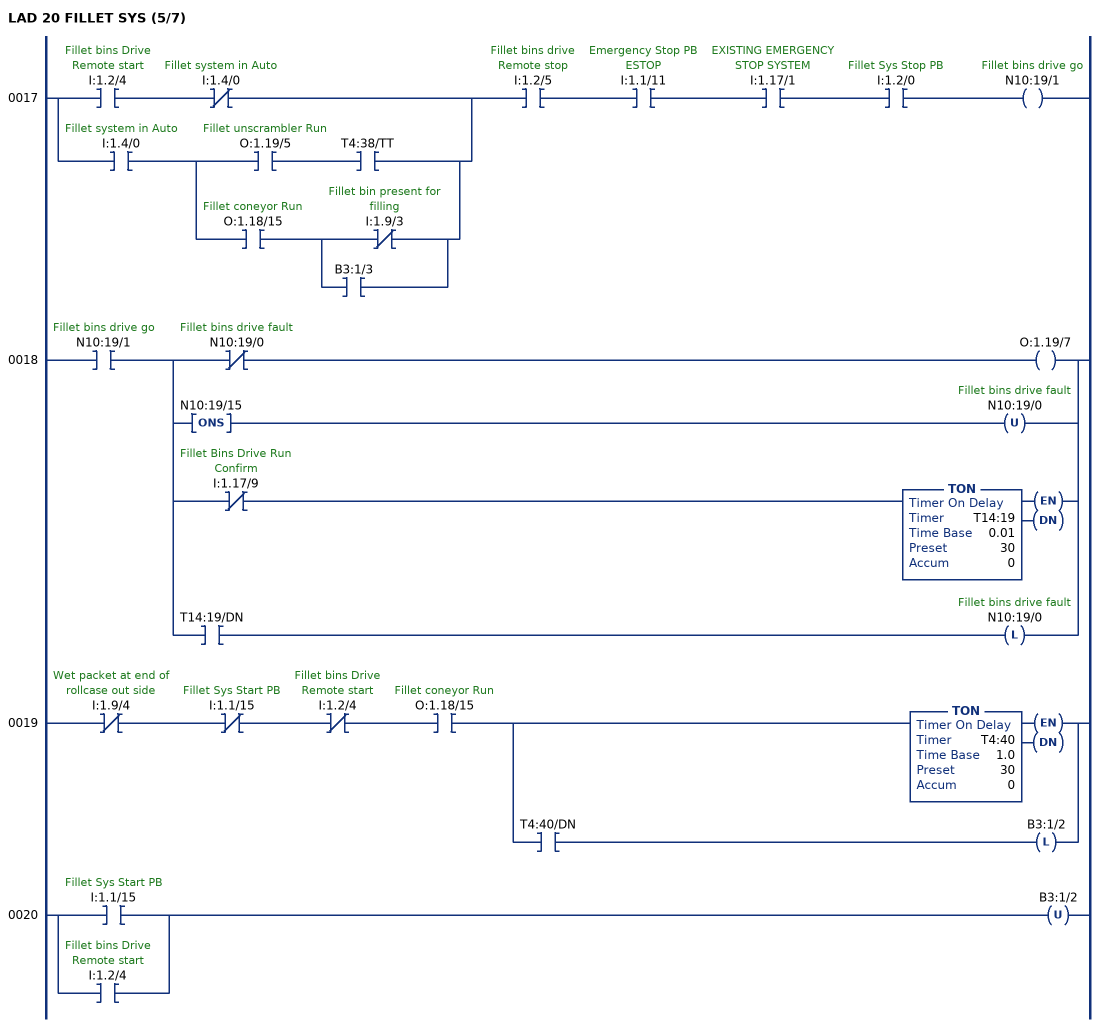
% Rung: 17 %
SOR BST XIC I:1.2/4 XIO I:1.4/0 NXB XIC I:1.4/0 BST XIC O:1.19/5 XIC T4:38/TT NXB XIC O:1.18/15 BST XIO I:1.9/3 NXB XIC B3:1/3 BND BND BND XIC I:1.2/5 XIC I:1.1/11 XIC I:1.17/1 XIC I:1.2/0 OTE N10:19/1 EOR
%   I:1.2/4  "Fillet bins Drive Remote start" %
%   I:1.4/0  "Fillet system in Auto" %
%   O:1.19/5  "Fillet unscrambler Run" %
%   O:1.18/15  "Fillet coneyor Run" %
%   I:1.9/3  "Fillet bin present for filling" %
%   I:1.2/5  "Fillet bins drive Remote stop" %
%   I:1.1/11  ESTOP  "Emergency Stop PB" %
%   I:1.17/1  "EXISTING EMERGENCY STOP SYSTEM" %
%   I:1.2/0  "Fillet Sys Stop PB" %
%   N10:19/1  "Fillet bins drive go" %
% Rung: 18 %
SOR XIC N10:19/1 BST XIO N10:19/0 OTE O:1.19/7 NXB OSR N10:19/15 OTU N10:19/0 NXB XIO I:1.17/9 TON T14:19 0.01 30 0 NXB XIC T14:19/DN OTL N10:19/0 BND EOR
%   N10:19/1  "Fillet bins drive go" %
%   N10:19/0  "Fillet bins drive fault" %
%   I:1.17/9  "Fillet Bins Drive Run Confirm" %
% Rung: 19 %
SOR XIO I:1.9/4 XIO I:1.1/15 XIO I:1.2/4 XIC O:1.18/15 BST TON T4:40 1.0 30 0 NXB XIC T4:40/DN OTL B3:1/2 BND EOR
%   I:1.9/4  "Wet packet at end of rollcase out side" %
%   I:1.1/15  "Fillet Sys Start PB" %
%   I:1.2/4  "Fillet bins Drive Remote start" %
%   O:1.18/15  "Fillet coneyor Run" %
% Rung: 20 %
SOR BST XIC I:1.1/15 NXB XIC I:1.2/4 BND OTU B3:1/2 EOR
%   I:1.1/15  "Fillet Sys Start PB" %
%   I:1.2/4  "Fillet bins Drive Remote start" %

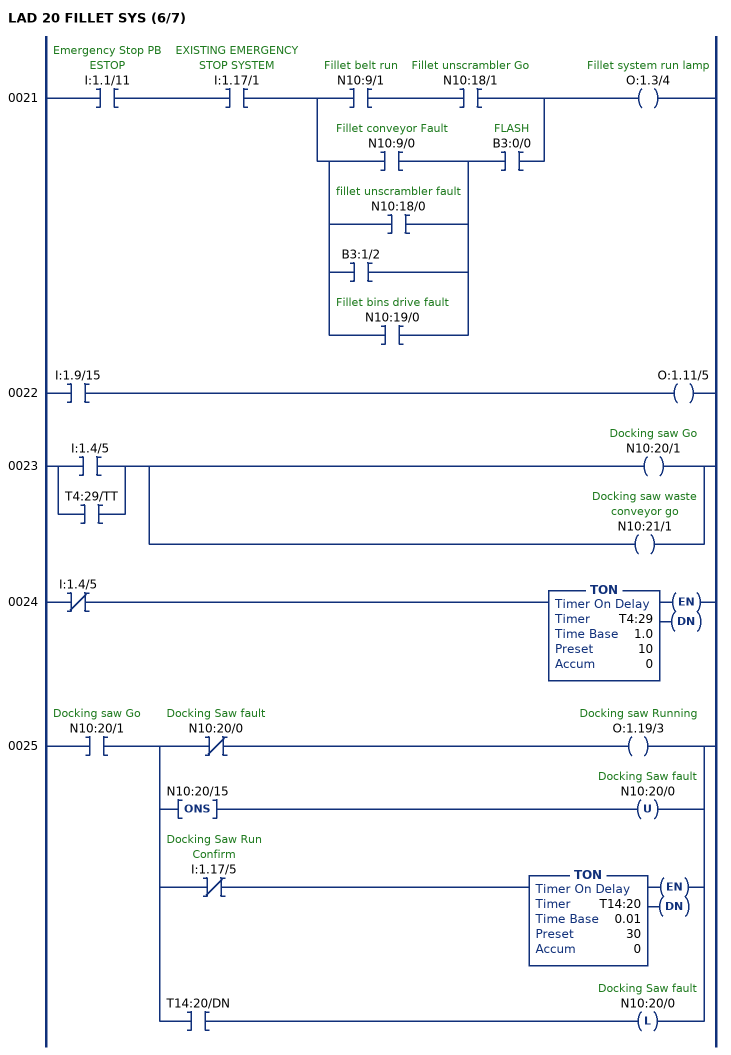
% Rung: 21 %
SOR XIC I:1.1/11 XIC I:1.17/1 BST XIC N10:9/1 XIC N10:18/1 NXB BST XIC N10:9/0 NXB XIC N10:18/0 NXB XIC B3:1/2 NXB XIC N10:19/0 BND XIC B3:0/0 BND OTE O:1.3/4 EOR
%   I:1.1/11  ESTOP  "Emergency Stop PB" %
%   I:1.17/1  "EXISTING EMERGENCY STOP SYSTEM" %
%   N10:9/1  "Fillet belt run" %
%   N10:18/1  "Fillet unscrambler Go" %
%   N10:9/0  "Fillet conveyor Fault" %
%   N10:18/0  "fillet unscrambler fault" %
%   N10:19/0  "Fillet bins drive fault" %
%   B3:0/0  FLASH %
%   O:1.3/4  "Fillet system run lamp" %
% Rung: 22 %
SOR XIC I:1.9/15 OTE O:1.11/5 EOR
% Rung: 23 %
SOR BST XIC I:1.4/5 NXB XIC T4:29/TT BND BST OTE N10:20/1 NXB OTE N10:21/1 BND EOR
%   N10:20/1  "Docking saw Go" %
%   N10:21/1  "Docking saw waste conveyor go" %
% Rung: 24 %
SOR XIO I:1.4/5 TON T4:29 1.0 10 0 EOR
% Rung: 25 %
SOR XIC N10:20/1 BST XIO N10:20/0 OTE O:1.19/3 NXB OSR N10:20/15 OTU N10:20/0 NXB XIO I:1.17/5 TON T14:20 0.01 30 0 NXB XIC T14:20/DN OTL N10:20/0 BND EOR
%   N10:20/1  "Docking saw Go" %
%   N10:20/0  "Docking Saw fault" %
%   O:1.19/3  "Docking saw Running" %
%   I:1.17/5  "Docking Saw Run Confirm" %

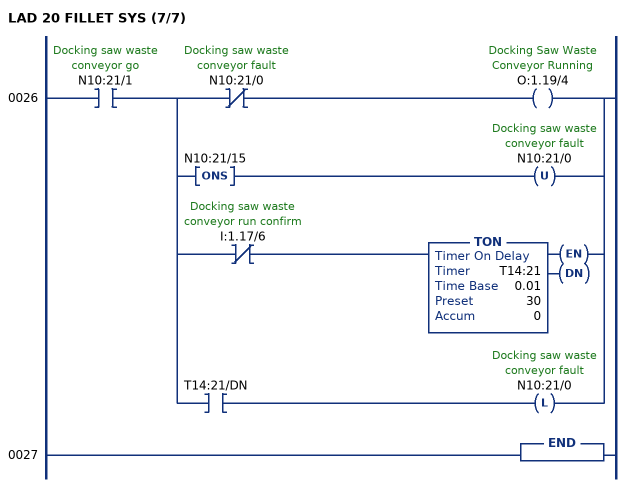
% Rung: 26 %
SOR XIC N10:21/1 BST XIO N10:21/0 OTE O:1.19/4 NXB OSR N10:21/15 OTU N10:21/0 NXB XIO I:1.17/6 TON T14:21 0.01 30 0 NXB XIC T14:21/DN OTL N10:21/0 BND EOR
%   N10:21/1  "Docking saw waste conveyor go" %
%   N10:21/0  "Docking saw waste conveyor fault" %
%   O:1.19/4  "Docking Saw Waste Conveyor Running" %
%   I:1.17/6  "Docking saw waste conveyor run confirm" %
% Rung: 27 %
SOR END EOR

OTHER DOCUMENTED ADDRESSES
    "t4"
  B3:2/3  "USE PREVIOUS LUG SPACE TIME"
  B3:3/0  "Dicky Stop Bit"
  B3:3/1  "Reset BTW on Error"
  B16:0/3  SURGE_DECK_RUNNING
  B16:0/10  "Temperary bit added as O:4/17 used twice in program suppect that existing output not reconfigured"
  C5:2  "BTW Error Counter"
  DFILE:0  "OUTPUT"
  DFILE:1  "INPUT"
  DFILE:2  "STATUS"
  DFILE:3  "BINARY"
  DFILE:4  "TIMER"
  DFILE:5  "COUNTER"
  DFILE:6  "CONTROL"
  DFILE:7  "INTEGER"
  DFILE:8  "FLOAT"
  I:1.8/2  "Deck 1 Tilthoist Detect PE"
  I:1.8/4  "Deck 1 Tilthoist ended limit switch"
  I:1.8/8  "Deck 1 Board Count"
  I:1.9/8  "Lug loader fiber photo eye"
  I:1.9/10  "Lug loader backlog photo eye"
  I:1.9/11  "Deck 1 board transfer Isolator"
  I:1.12/12  "Isolator Auxillary M1534"
  I:1.12/13  "Isolator Auxillary M1535"
  I:1.12/14  "Isolator Auxillary M1536"
  I:1.12/15  "Isolator Auxillary M1537"
  I:2.0/9  "Deck 1 VSD Fault"
  I:3.0/14  "Deck 1 board transfer run confirm"
  I:3.0/15  "Round table Run confirm"
  M00000:002.001/01  "Outputs Enabled"
  M00000:002.001/02  "Counter Hold"
  M00000:002.001/03  "Counter Decrement"
  M00000:002.001/04  "Counter Reset"
  M00000:002.001/05  "Bit 1 Reset Mode"
  M00000:002.001/06  "Bit 2 Reset Mode"
  M00000:002.001/07  "Bit 3 Reset Mode"
  M00000:002.001/09  "Bit 1 Input Type"
  M00000:002.001/10  "Bit 2 Input Type"
  M00000:002.001/11  "Bit 3 Input Type"
  M00000:002.001/12  "Enable Counter"
  M00000:002.001/13  "Counter Ring"
  M00000:002.001/14  "Bit 1 Operating Mode"
  M00000:002.001/15  "Bit 2 Operating Mode"
  M00000:002.009  "Rate Period"
  M00000:002.034  "Maximum count value"
  MOV  
  N7:1  "LUG SPACE TIME"
  N7:5  "TIME FOR THE LAST LUG SPACE WITH NO SPEED CHANGES, USED WHEN THERE HAS BEEN A SLOW DOWN"
  N7:6  "LUG LOADER LOAD DELAY"
  N7:7  "LUGS PER MIN"
  N7:26  "TIME VALUE USED WHEN CHAINS ARE RUNNING SLOW TO CUT BOARD IN SAW"
  N7:27  N7  "OFF DELAY FOR MANUAL WET BOARD MARKING LIGHT, 0-10 LUG SPACES"
  N7:64/15  "VIRTUAL BTW ENABLE BIT"
  N9:1  "Remote Chassis Slot 5 Word 1"
  N9:2  "Remote Chassis Slot 5 Word 2"
  N10:1  "Deck 1 Pkt Conv A FWD"
  N10:8/0  "Deck 1 Board transfer Fault"
  N10:10/0  "Fillet table fault"
  N10:15/1  "Deck 2 Board tarnsfer run"
  O:1.10/5  "Deck 1 Ducker down signal"
  O:1.11/1  "Deck 1timber stops up signal"
  O:4.16  "LUg Loader Backlog Deck Run"
  O:5.1  "Deck1 board transfer #2 speed"
  O:5.2  "Deck1 board transfer #3 speed"
  T4:0  "Flasher timer"
  T4:24  "Lug Loader Lug Period Timer"
  T4:33  "VIRTUAL LUG SPACE TIME"

COMMENTS NOT ATTACHED TO A CURRENT RUNG
  O:4.0/8: Run lamp for deck 1 board transfer 1
  RUNG000005-000019: MARK WET BOARDS WITH PAINT.
  RUNG000005-000020: THE NEXT 2 RUNGS ARE FOR PUTTING A 2 INTO TO THE SHIFT REGISTER TO REPRESENT THAT THE BOARD WAS WET. THE MOISTURE METER IS ON THE ZERO MARK OF THE TIMING, THIS WAS CAUSING  SOME PROBLEMS WITH DROPPING OUT THE CORRECT BOARD, AS SOMETIMES THE 2 WAS GETTING PUT IN THE WRONG LUG SPACE, TO GET AROUND THIS THERE IS NOW A DELAY OF 3/10TH OF A LUG SPACE BEFORE THE 2 IS PUT IN
  RUNG000005-000024: DROP OUT GATE DOWN
  RUNG000005-000025: DROP OUT GATE UP
  RUNG000005-000028: THESE NEXT 2 RUNGS ARE FOR THE PE CLEANING AIR BLOWERS ON THE LUGLOADER AND THE MOISTURE METER. THE 1ST ONE IS THE INTERVAL TIMER AND THE 2ND IS THE AIR ON TIME

REVISION NOTES
  0: Upgraded Processor, Added new RIO rack and ASB - 3-1-07

DATA TABLE (non-zero values as saved)
DATA B3
% B3:0 % 0X4000 0X4140 0X000A 0X0002 0X0000 0X0000 0X0000 0X0000 0X0000 0X0000
% B3:10 % 0XC000 0X0000 0X0000 0X0000 0X0000 0X0002 0X0000 0X0000 0X0000 0X0000
DATA T4
% .PRE .ACC %
% T4:0 % 2000 0
% T4:1 % 5 5
% T4:2 % 5 5
% T4:3 % 5 5
% T4:4 % 5 5
% T4:5 % 2 2
% T4:6 % 2 2
% T4:7 % 15 0
% T4:8 % 13 0
% T4:9 % 30 30
% T4:10 % 100 0
% T4:11 % 50 0
% T4:12 % 3 3
% T4:13 % 60 60
% T4:14 % 40 0
% T4:15 % 250 0
% T4:16 % 1 1
% T4:17 % 50 50
% T4:18 % 5 0
% T4:19 % 3 3
% T4:20 % 3 3
% T4:21 % 4 4
% T4:22 % 5 5
% T4:23 % 6 1
% T4:24 % 500 322
% T4:25 % 100 0
% T4:26 % 20 0
% T4:27 % 300 0
% T4:28 % 18 0
% T4:29 % 10 0
% T4:30 % 150 0
% T4:31 % 10 0
% T4:32 % 40 0
% T4:33 % 50 0
% T4:34 % 5 0
% T4:35 % 5 0
% T4:36 % 10 8
% T4:37 % 600 0
% T4:38 % 20 0
% T4:39 % 100 0
% T4:40 % 30 0
% T4:41 % 10 10
% T4:42 % 20 20
% T4:43 % 2 0
% T4:44 % 4 0
% T4:45 % 18 0
% T4:46 % 15 0
% T4:47 % 100 100
% T4:48 % 17 0
% T4:49 % 20 0
% T4:50 % 1000 0
% T4:52 % 9 0
% T4:53 % 10 0
% T4:54 % 3 0
% T4:55 % 40 0
DATA C5
% .PRE .ACC %
% C5:0 % 100 8
% C5:1 % 100 6
% C5:2 % 30000 349
% C5:3 % 5 3
% C5:4 % 4 420
% C5:10 % 30000 10
DATA R6
% .LEN .POS %
% R6:0 % 20 0
DATA N7
% N7:0 % 6000 500 7900 5001 7900 500 6 12 6 5
% N7:10 % 1 1 1 1 1 1 1 1 1 1
% N7:20 % 1 1 1 1 1 1 450 0 0 0
% N7:30 % 1 1 1 1 1 1 1 1 1 1
% N7:40 % 1 1 1 1 1 0 0 0 0 0
% N7:50 % -32768 0 0 17408 0 0 0 -9 0 0
% N7:90 % 0 1200 1900 1999 2000 2100 0 0 0 0
DATA F8
% F8:0 % 11100
DATA N9
% N9:0 % 7900 0 0 6000 0 0 0 0 0 0
% N9:10 % -15320 4 0 0 0 0 0 0 0 0
DATA N10
% N10:0 % 0 0 0 0 0 0 0 -32766 0 0
% N10:10 % -32767 0 0 0 0 0 -32766 0 0 0
% N10:20 % -32766 -32766 -32766 -32762 -32765 0 0 0 0 0
DATA N11
% N11:0 % 3326 25 960 1100 23 0 0 1 1 14689
% N11:10 % -31743 0 90 40 0 0 0 100 0 0
% N11:20 % 0 100 40 10 89 1 2 0 0 3
% N11:30 % -27264 2053 90 0 0 256 90 0 0 0
% N11:50 % 32767 0 0 0 0 0 0 0 0 0
DATA T12
% .PRE .ACC %
% T12:0 % 1000 1001
% T12:1 % 200 0
% T12:2 % 500 185
% T12:3 % 14 24
% T12:4 % 15 7
DATA N13
% N13:0 % 32 27712 1 32 0 0 0 0 0 50
% N13:10 % 400 0 0 0 0 0 0 0 0 0
% N13:30 % 0 0 0 0 3332 0 0 0 0 0
DATA T14
% .PRE .ACC %
% T14:1 % 30 0
% T14:2 % 30 0
% T14:3 % 30 0
% T14:4 % 30 0
% T14:5 % 30 0
% T14:6 % 30 0
% T14:7 % 50 0
% T14:8 % 30 0
% T14:9 % 30 0
% T14:10 % 30 0
% T14:11 % 30 0
% T14:12 % 30 0
% T14:13 % 30 0
% T14:14 % 30 0
% T14:16 % 30 0
% T14:17 % 30 0
% T14:18 % 30 0
% T14:19 % 30 0
% T14:20 % 30 0
% T14:21 % 30 0
% T14:22 % 25 0
% T14:23 % 300 0
% T14:24 % 3 3
% T14:25 % 3 3
% T14:26 % 2000 0
DATA C15
% .PRE .ACC %
% C15:0 % 100 1
% C15:1 % 100 0
DATA B16
% B16:0 % 0X0002 0X0000 0X0000 0X0000 0X0000 0X0000 0X0000 0X0000 0X0000 0X0000
